// TIA Portal V17 export
// export: Created 2022-05-07T16:38:47.0736851Z, ExportSetting WithDefaults, DisplayName Totally Integrated Automation Portal, DisplayVersion V17 Update 3, DisplayName TIA Portal Openness, DisplayVersion V17 Update 3, DisplayName TIA Portal Version Control Interface, DisplayVersion V17, DisplayName TIA Portal Test Suite Advanced, DisplayVersion V17 Update 1, DisplayName SINAMICS Startdrive Advanced, DisplayVersion V17 Update2, DisplayName SINAMICS Startdrive G130, G150, S120, S150, SINAMICS MV, S210, DisplayVersion V17 Update2, DisplayName SINAMICS Startdrive G110M, G120, G120C, G120D, G120P, G115D, DisplayVersion V17 Update2, DisplayName STEP 7 Professional, DisplayVersion V17 Update 3, DisplayName STEP 7 Safety, DisplayVersion V17, DisplayName WinCC UA Professional, DisplayVersion V17 Update 3
FUNCTION_BLOCK "ALLARMI"   // FB13, LAD
TITLE = COMPILAZIONE ALLARMI HMI
{ S7_Optimized_Access := 'TRUE' }
VERSION : 0.1
// stored: AutoNumber true, IsIECCheckEnabled false, IsRetainMemResEnabled false, MemoryReserve 100, SetENOAutomatically false, UDAEnableTagReadback false
BEGIN

REGION Network 1: ALLA HOMING MS
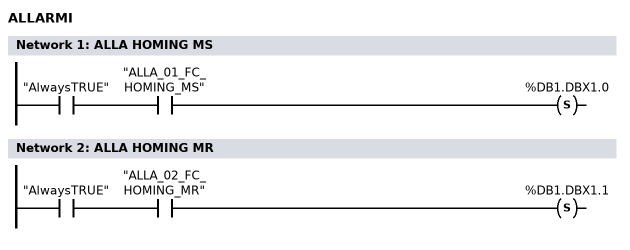
   RUNG wire#powerrail
      Contact( "AlwaysTRUE" )
      Contact( "ALLA_01_FC_HOMING_MS" )
      S_Coil( %DB1.DBX1.0 )
   END_RUNG
   // the same network as SCL:
   IF "AlwaysTRUE" AND "ALLA_01_FC_HOMING_MS" THEN %DB1.DBX1.0 := TRUE; END_IF;
END_REGION

REGION Network 2: ALLA HOMING MR
   RUNG wire#powerrail
      Contact( "AlwaysTRUE" )
      Contact( "ALLA_02_FC_HOMING_MR" )
      S_Coil( %DB1.DBX1.1 )
   END_RUNG
   // the same network as SCL:
   IF "AlwaysTRUE" AND "ALLA_02_FC_HOMING_MR" THEN %DB1.DBX1.1 := TRUE; END_IF;
END_REGION
END_FUNCTION_BLOCK
